// TIA Portal project "BasculeBridgeS7_1200" (V15.1)

(* hardware
DEVICE "S7-1200-Station_1"  S7-1200 Station
   slot 0: "Baugruppenträger_0"  S7-1200 Rack  Rack  V1.0
   slot 1: "PLC_1"  CPU 1212C DC/DC/DC  6ES7 212-1AE40-0XB0  V4.2
   slot 2: "AQ 2x14BIT_1"  6ES7 232-4HB30-0XB0  V1.0
*)

// ===== PLC "PLC_1"  CPU 1212C DC/DC/DC =====

VAR_GLOBAL   // PLC tag table "Standard-Variablentabelle"
   "FlagControlOn" AT %M0.0 : Bool;
   "FlagOpenMonitoringTimeError" AT %M0.1 : Bool;
   "FlagCloseMonitoringTimeError" AT %M0.2 : Bool;
   "S5ResetMovementError" AT %E0.6 : Bool;
   "ElapsedMonitoringTimeOpen" AT %AW10 : Int;
   "ElapsedMonitoringTimeClose" AT %AW12 : Int;
END_VAR

VAR_GLOBAL   // PLC tag table "Variablentabelle aus XML_1"
   "M1Open" AT %Q0.0 : Bool;
   "M1Close" AT %Q0.1 : Bool;
   "P1IsOpen" AT %Q0.2 : Bool;
   "P2IsClosed" AT %Q0.3 : Bool;
   "ErrorWhileMovement" AT %Q0.4 : Bool;
   "S1ControlOn" AT %I0.0 : Bool;
   "S2ControlOff" AT %I0.1 : Bool;   // NC
   "S3OpenBridge" AT %I0.2 : Bool;
   "S4CloseBridge" AT %I0.3 : Bool;
   "B1BridgeIsClosed" AT %I0.4 : Bool;
   "B2BridgeIsOpen" AT %I0.5 : Bool;
   "P3ControlOn" AT %Q0.5 : Bool;
END_VAR

// folder: System blocks/Program resources

DATA_BLOCK "IEC_Timer_Open_DB"   // DB1
{ S7_Optimized_Access := 'TRUE' }
AUTHOR : Simatic
FAMILY : IEC
NAME : IEC_TMR
VERSION : 1.0
// stored: InstanceOfName IEC_TIMER
"IEC_TIMER"
BEGIN
END_DATA_BLOCK

DATA_BLOCK "IEC_Timer_Close_DB"   // DB2
{ S7_Optimized_Access := 'TRUE' }
AUTHOR : Simatic
FAMILY : IEC
NAME : IEC_TMR
VERSION : 1.0
// stored: InstanceOfName IEC_TIMER
"IEC_TIMER"
BEGIN
END_DATA_BLOCK

// folder: (top level)

FUNCTION "MHJ-PLC-Lab-Function-S71200" : Void   // FC9000, SCL
{ S7_Optimized_Access := 'TRUE' }
VERSION : 0.1
   VAR_TEMP
      rdTimeReturn : Int;
      outputTime : DTL;
      SyncVal : Byte;
      forVal : Int;
      forVal_2 : Int;
      Value : Byte;
   END_VAR
   VAR CONSTANT
      CompVal : Byte := 16#34;
      Value_01 : Byte := 16#11;
      Value_01_DW : DWord := 16#A165_D992;
      Value_02_DW : DWord := 16#58BE_4401;
   END_VAR
BEGIN

   #Value:=PEEK(area := 16#82,
        dbNumber := 0,
        byteOffset := 511);
   #Value := #Value + 1;

   POKE(area := 16#82,
        dbNumber := 0,
        byteOffset := 511,
        value := #Value);

   POKE(area:=16#81,
        dbNumber:=0,
        byteOffset:=1016,
        value:=#Value_01_DW);
   POKE(area := 16#81,
        dbNumber := 0,
        byteOffset := 1020,
        value := #Value_02_DW);

   POKE(area := 16#81,
        dbNumber := 0,
        byteOffset := 511,
        value := B#16#00);

   FOR #forVal := 0 TO 120 DO
       FOR #forVal_2:=0 TO 10 DO
           #rdTimeReturn:=RD_SYS_T(#outputTime);
           #rdTimeReturn := WR_SYS_T(#outputTime);
           #rdTimeReturn := RD_SYS_T(#outputTime);
           #rdTimeReturn := WR_SYS_T(#outputTime);
       END_FOR;
       #SyncVal:= PEEK(area := 16#81,
                      dbNumber := 0,
                      byteOffset := 511);
       IF #SyncVal = #CompVal THEN
          GOTO M_1;
       END_IF;
   END_FOR;
   RETURN;

   M_1:
   POKE(area := 16#81,
        dbNumber := 0,
        byteOffset := 511,
        value := B#16#0);
END_FUNCTION

ORGANIZATION_BLOCK "Main"   // OB1, FBD, ProgramCycle
TITLE = "Main Program Sweep (Cycle)"
{ S7_Optimized_Access := 'TRUE' }
VERSION : 0.1
   VAR_INPUT
      Initial_Call : Bool;   // Initial call of this OB
      Remanence : Bool;   // =True, if remanent data are available
   END_VAR
BEGIN

REGION Network 1
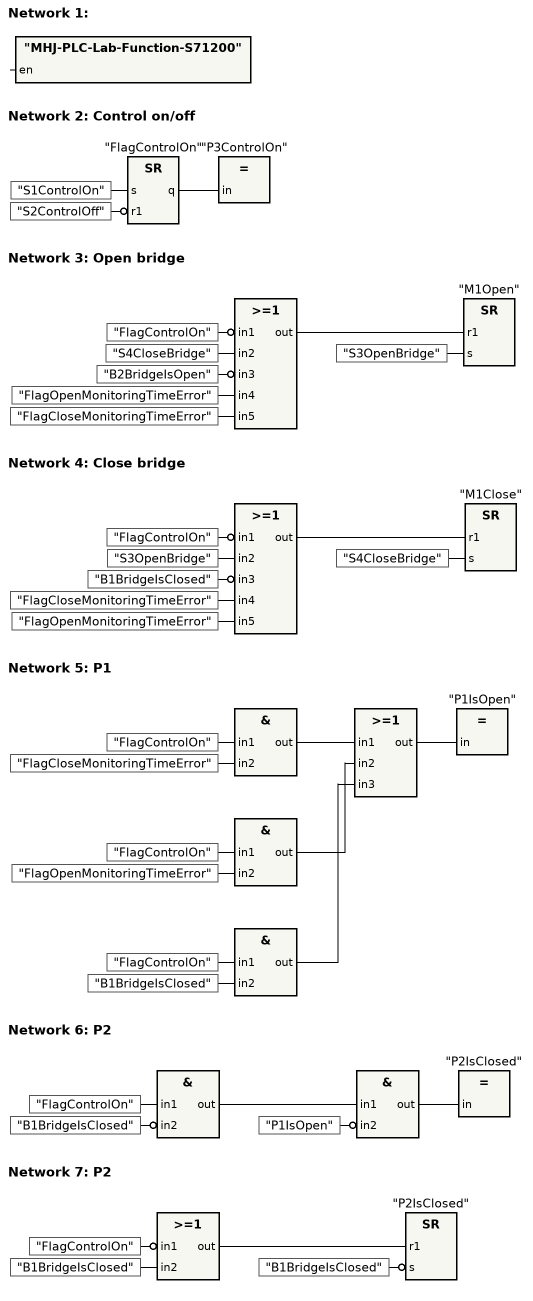
   "MHJ-PLC-Lab-Function-S71200"();
END_REGION

REGION Network 2: Control on/off
   IF "S1ControlOn" THEN
       "FlagControlOn" := TRUE;   // SR flip-flop
   END_IF;
   IF NOT "S2ControlOff" THEN "FlagControlOn" := FALSE; END_IF;
   "P3ControlOn" := "FlagControlOn";
END_REGION

REGION Network 3: Open bridge
   IF "S3OpenBridge" THEN
       "M1Open" := TRUE;   // SR flip-flop
   END_IF;
   IF NOT "FlagControlOn" OR "S4CloseBridge" OR NOT "B2BridgeIsOpen" OR "FlagOpenMonitoringTimeError" OR "FlagCloseMonitoringTimeError" THEN
       "M1Open" := FALSE;
   END_IF;
END_REGION

REGION Network 4: Close bridge
   IF "S4CloseBridge" THEN
       "M1Close" := TRUE;   // SR flip-flop
   END_IF;
   IF NOT "FlagControlOn" OR "S3OpenBridge" OR NOT "B1BridgeIsClosed" OR "FlagCloseMonitoringTimeError" OR "FlagOpenMonitoringTimeError" THEN
       "M1Close" := FALSE;
   END_IF;
END_REGION

REGION Network 5: P1
   "P1IsOpen" := ("FlagControlOn" AND "FlagCloseMonitoringTimeError") OR ("FlagControlOn" AND "FlagOpenMonitoringTimeError") OR ("FlagControlOn" AND "B1BridgeIsClosed");
END_REGION

REGION Network 6: P2
   "P2IsClosed" := "FlagControlOn" AND NOT "B1BridgeIsClosed" AND NOT "P1IsOpen";
END_REGION

REGION Network 7: P2
   IF NOT "B1BridgeIsClosed" THEN
       "P2IsClosed" := TRUE;   // SR flip-flop
   END_IF;
   IF NOT "FlagControlOn" OR "B1BridgeIsClosed" THEN "P2IsClosed" := FALSE; END_IF;
END_REGION

REGION Network 8: Open monitoring time
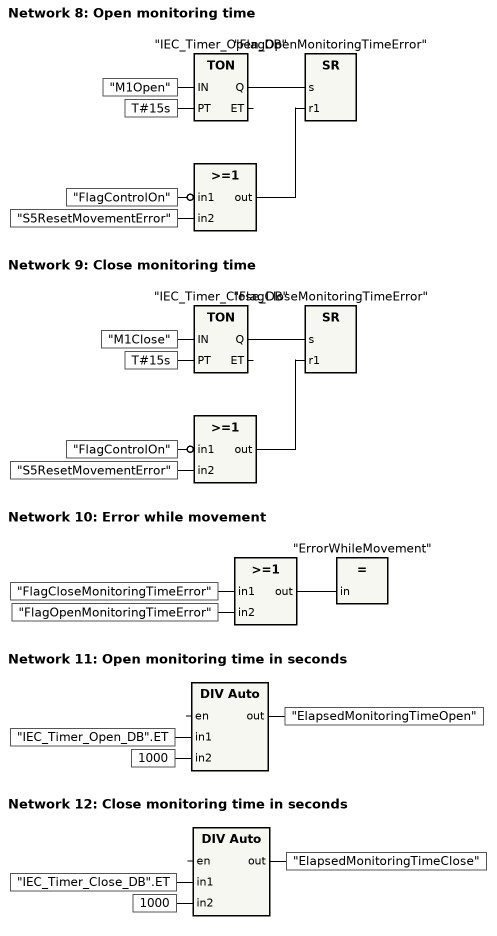
   "IEC_Timer_Open_DB".TON(IN := "M1Open", PT := T#15s);
   IF "IEC_Timer_Open_DB".Q THEN
       "FlagOpenMonitoringTimeError" := TRUE;   // SR flip-flop
   END_IF;
   IF NOT "FlagControlOn" OR "S5ResetMovementError" THEN "FlagOpenMonitoringTimeError" := FALSE; END_IF;
END_REGION

REGION Network 9: Close monitoring time
   "IEC_Timer_Close_DB".TON(IN := "M1Close", PT := T#15s);
   IF "IEC_Timer_Close_DB".Q THEN
       "FlagCloseMonitoringTimeError" := TRUE;   // SR flip-flop
   END_IF;
   IF NOT "FlagControlOn" OR "S5ResetMovementError" THEN "FlagCloseMonitoringTimeError" := FALSE; END_IF;
END_REGION

REGION Network 10: Error while movement
   "ErrorWhileMovement" := "FlagCloseMonitoringTimeError" OR "FlagOpenMonitoringTimeError";
END_REGION

REGION Network 11: Open monitoring time in seconds
   "ElapsedMonitoringTimeOpen" := "IEC_Timer_Open_DB".ET / 1000;
END_REGION

REGION Network 12: Close monitoring time in seconds
   "ElapsedMonitoringTimeClose" := "IEC_Timer_Close_DB".ET / 1000;
END_REGION
END_ORGANIZATION_BLOCK